// TIA Portal V20 export
FUNCTION "FIT100" : Void   // FC4, FBD
{ S7_Optimized_Access := 'TRUE' }
// stored: SetENOAutomatically false
   VAR_TEMP
      Temp : "DigVal";
      Temp_1 : "DigVal";
   END_VAR
BEGIN

REGION Network 1: Channel input
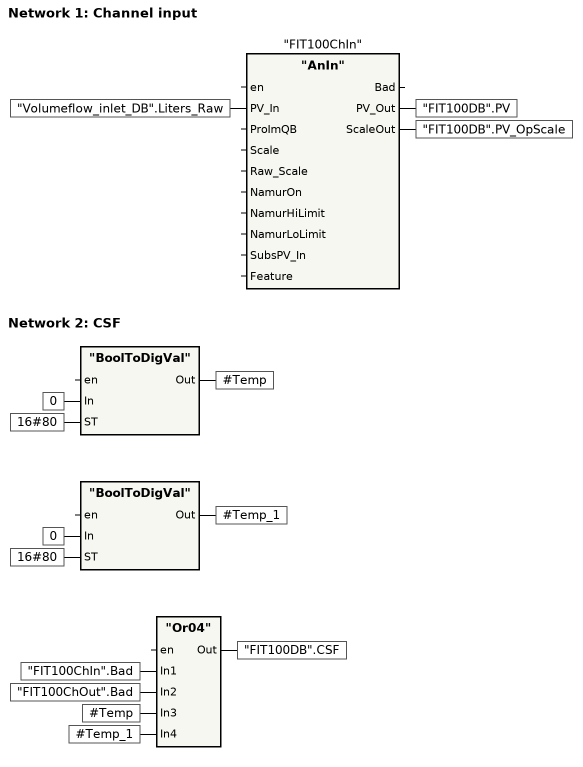
   "FIT100ChIn"(PV_In := "Volumeflow_inlet_DB".Liters_Raw,   // "AnIn"
                PV_Out => "FIT100DB".PV,
                ScaleOut => "FIT100DB".PV_OpScale);
END_REGION

REGION Network 2: CSF
   "BoolToDigVal"(In := 0, ST := 16#80, Out => #Temp);
   "BoolToDigVal"(In := 0, ST := 16#80, Out => #Temp_1);
   "Or04"(In1 := "FIT100ChIn".Bad,
          In2 := "FIT100ChOut".Bad,
          In3 := #Temp,
          In4 := #Temp_1,
          Out => "FIT100DB".CSF);
END_REGION

REGION Network 3: MonAnL
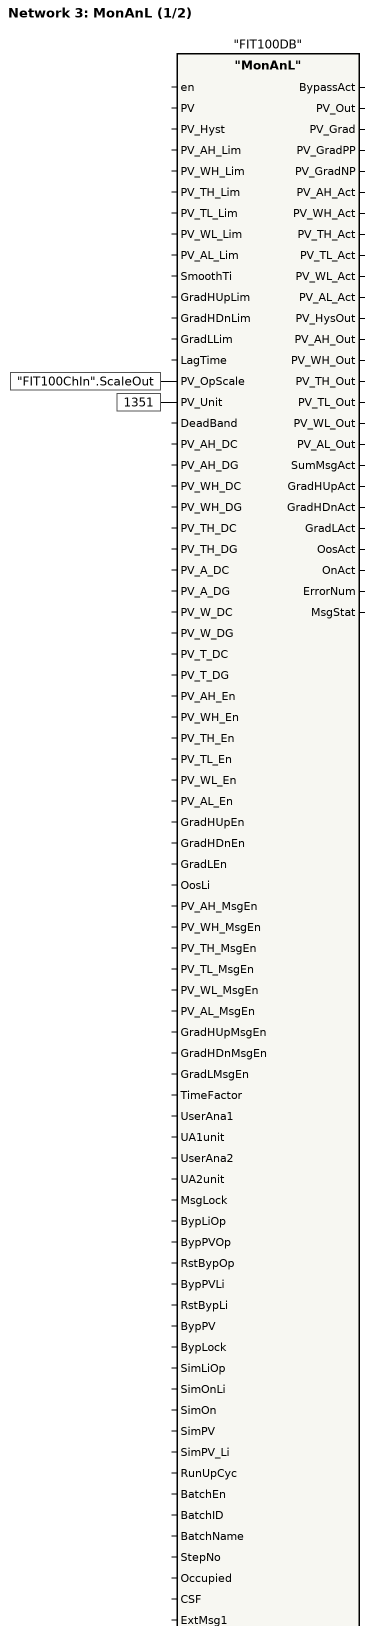
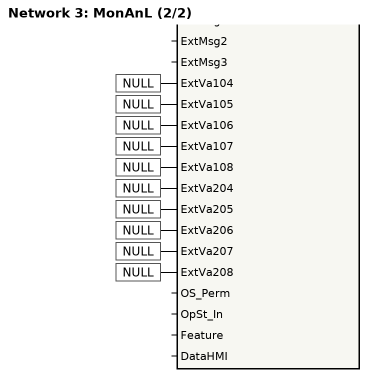
   "FIT100DB"(PV_OpScale := "FIT100ChIn".ScaleOut,   // "MonAnL"
              PV_Unit := 1351,
              ExtVa104 := NULL,
              ExtVa105 := NULL,
              ExtVa106 := NULL,
              ExtVa107 := NULL,
              ExtVa108 := NULL,
              ExtVa204 := NULL,
              ExtVa205 := NULL,
              ExtVa206 := NULL,
              ExtVa207 := NULL,
              ExtVa208 := NULL);
END_REGION

REGION Network 4: MTP
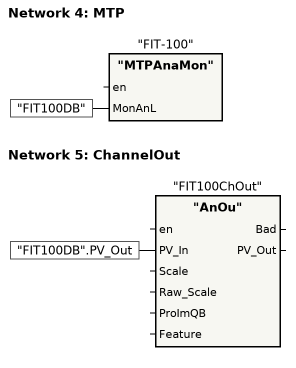
   "FIT-100"(MonAnL := "FIT100DB");   // "MTPAnaMon"
END_REGION

REGION Network 5: ChannelOut
   "FIT100ChOut"(PV_In := "FIT100DB".PV_Out);   // "AnOu"
END_REGION
END_FUNCTION
